(* IEC 61131-3 sources: CodesysTest/export/UN00 - Sharp Bagger/EM01 - Bagger Head/CM03 - Sealer/Pneumatic/FB_PneumaticSealer.pou, 1 file *)

(* ---- FB_PneumaticSealer.pou.st ---- *)
(*#-#-#-#-#-#-#-#-#-#---Declaration---#-#-#-#-#-#-#-#-#-#-#-#-#*)

FUNCTION_BLOCK FINAL FB_PneumaticSealer EXTENDS FB_BasicSealer
VAR_INPUT
	cylinder : ICylinder;
END_VAR
VAR_OUTPUT
END_VAR
VAR

END_VAR
(*#-#-#-#-#-#-#-#-#-#---Implementation---#-#-#-#-#-#-#-#-#-#-#-#-#*)

SUPER^();

EnableSimulation(cylinder,simulateIO);

IF sealActive THEN
	cylinder.Extend();
ELSE
	cylinder.Retract();
END_IF
